FUNCTION_BLOCK FB_InputDebounce
VAR_INPUT
	I	: typFBDInput;
END_VAR

VAR_IN_OUT
	IQ	: typFBDInOut;
END_VAR

VAR_OUTPUT
	Q	: typFBDOutput;
END_VAR

VAR
	tonOnDelay		: TON;
	tofOffDelay		: TOF;
	uiDebounceSM	: UINT;
END_VAR

tonOnDelay(PT	:= I.tOnDelay);
tofOffDelay(PT	:= I.tOffDelay);

CASE uiDebounceSM OF
	
0: // If there is a trig, then set a timer for the On Delay
IF IQ.xTrig THEN
	tonOnDelay.IN	:= TRUE;
	tofOffDelay.IN	:= TRUE;
	uiDebounceSM	:= 10;
END_IF

10: // If timer is completed, set the timer false, set the Gate (output) high, falling edge to TOF input
IF tonOnDelay.Q THEN
	tonOnDelay.IN	:= FALSE;
	Q.xGate			:= TRUE;
	tofOffDelay.IN	:= FALSE;
	uiDebounceSM	:= 20;	
END_IF

20: // Falling edge on TOF drops Gate
IF NOT tofOffDelay.Q AND NOT IQ.xTrig THEN
	Q.xGate			:= FALSE;
	uiDebounceSM	:= 30;
ELSIF NOT tofOffDelay.Q AND IQ.xTrig THEN
//Jump state; no other actions (do not set gate false)
	uiDebounceSM	:= 40;
END_IF

30: //Ensure the trig has gone low
IF NOT IQ.xTrig THEN
	uiDebounceSM	:= 0;
END_IF

40: // State for "if trig held past OffDelay time"; if trig has gone low, set gate low
IF NOT IQ.xTrig THEN
	Q.xGate			:= FALSE;
	uiDebounceSM	:= 0;
END_IF
	
END_CASE

END_FUNCTION_BLOCK

(* stored: Version 1.1.0.1, ProductVersion 3.1.4024.6
   POU FB_InputDebounce: Id {a5a2ec82-c70f-4302-80ec-2dc51ff0b611}, SpecialFunc None *)
